TYPE "A0301_Mach_Ax_Pos_Data"
VERSION : 0.1
// Block: A0301_Mach_Ax_Pos_Data
   STRUCT
      OffsetPosAttesa : LReal;
      PosAttesa : LReal;
      PosFineSpinta : LReal;
   END_STRUCT;

END_TYPE
